// Mitsubishi GX Works2 project: group10   PLC: FX3G

// global labels: Global1
VAR_GLOBAL
  EmergencyEnd AT X005 : BOOL;
  EndDay AT M7 : BOOL;
  MaterialMissing AT M6 : BOOL;
  WorkDayActive AT Y007 : BOOL;
  PrepStart AT X001 : BOOL;
  AnalogInput1 AT D8280 : INT;
  FloatInput AT D6000 : REAL;
END_VAR
VAR_GLOBAL CONSTANT
  Constant400 : REAL := E400.0;
END_VAR
VAR_GLOBAL
  TypeValue AT D1900 : REAL;
END_VAR
VAR_GLOBAL CONSTANT
  Const6 : REAL := 6.0;
END_VAR
VAR_GLOBAL
  Pinuk AT M2 : BOOL;
END_VAR
VAR_GLOBAL CONSTANT
  Const5 : REAL := 5.0;
END_VAR
VAR_GLOBAL
  Ragil AT M3 : BOOL;
  KeepPinuk AT M10 : BOOL;
  KeepRagil AT M12 : BOOL;
  InputRaspberryAmount AT D1500 : REAL;
  RaspberryAmount AT D1510 : REAL;
  InputLemonAmount AT D1600 : REAL;
  LemonAmount AT D1610 : REAL;
  InputMaterialAmount AT D1700 : REAL;
  MaterialAmount AT D1710 : REAL;
  InputGummyAmount AT D1800 : REAL;
  GummyAmount AT D1810 : REAL;
END_VAR
VAR_GLOBAL CONSTANT
  MinRaspberryPinuk : REAL := 385.0;
  MinLemonPinuk : REAL := 665.0;
  MinMaterialPinuk : REAL := 210.0;
  MinGummyPinuk : REAL := 70.0;
END_VAR
VAR_GLOBAL
  CantMakePinuk AT M13 : BOOL;
END_VAR
VAR_GLOBAL CONSTANT
  MinRaspberryRagil : REAL := 280.0;
  MinLemonRagil : REAL := 455;
  MinMaterialRagil : REAL := 105;
  MinGummyRagil : REAL := 28;
END_VAR
VAR_GLOBAL
  CantMakeRagil AT M14 : BOOL;
  StartWorkDay AT X007 : BOOL;
  Invalid AT M77 : BOOL;
  StartMaking AT M8 : BOOL;
END_VAR
VAR_GLOBAL CONSTANT
  Const0 : REAL := E0.0;
  Const700 : REAL := E700.0;
END_VAR
VAR_GLOBAL
  ContainerMR AT D1400 : REAL;
END_VAR
VAR_GLOBAL CONSTANT
  Const560 : REAL := E560.0;
END_VAR
VAR_GLOBAL
  ContainerML AT D1300 : REAL;
END_VAR
VAR_GLOBAL CONSTANT
  Const490 : REAL := E490.0;
  Const350 : REAL := E350.0;
END_VAR
VAR_GLOBAL
  HoldTime AT M9 : BOOL;
  TC_1 AT TC1 : BOOL;
END_VAR
VAR_GLOBAL CONSTANT
  Const5sec : INT := 50;
END_VAR
VAR_GLOBAL
  EndMakingLight AT TS1 : BOOL;
  Making AT Y000 : BOOL;
  Freezing AT X002 : BOOL;
  TempS AT X003 : BOOL;
  FinishFreezing AT TS2 : BOOL;
  FreezingLight AT Y002 : BOOL;
  TC_2 AT TC2 : BOOL;
END_VAR
VAR_GLOBAL CONSTANT
  Const8sec : INT := 80;
END_VAR
VAR_GLOBAL
  ContainerFL AT D1310 : REAL;
  ContainerFR AT D1410 : REAL;
  Mixing AT M15 : BOOL;
  ContainerMix AT D1955 : REAL;
  PinukMixed AT M20 : BOOL;
  RagilMixed AT M30 : BOOL;
  TimerMixPinuk AT TC10 : BOOL;
END_VAR
VAR_GLOBAL CONSTANT
  Mix5Sec : INT := 50;
END_VAR
VAR_GLOBAL
  StopMixPinuk AT TS10 : BOOL;
  FinishMixPinukLight AT M40 : BOOL;
  TimerMixRagil AT TC11 : BOOL;
END_VAR
VAR_GLOBAL CONSTANT
  Mix3Sec : INT := 30;
END_VAR
VAR_GLOBAL
  StopMixRagil AT TS11 : BOOL;
  FinishMixRagilLight AT M50 : BOOL;
  HelpFlick AT M60 : BOOL;
  TC_3 AT TC3 : BOOL;
  HelpFlick1 AT TS3 : BOOL;
  Flick1 AT Y005 : BOOL;
  TC_4 AT TC4 : BOOL;
  HelpFlick2 AT TS4 : BOOL;
  Flick2 AT Y006 : BOOL;
END_VAR
VAR_GLOBAL CONSTANT
  Const1Sec : INT := 10;
END_VAR
VAR_GLOBAL
  PackageAmount AT D1360 : REAL;
END_VAR
VAR_GLOBAL CONSTANT
  AddOnePackage : REAL := 1;
  Const40 : REAL := E40.0;
END_VAR
VAR_GLOBAL
  OutputP AT D1100 : REAL;
  AnalogOutput AT D8282 : INT;
  WaitToPack AT M90 : BOOL;
END_VAR

// task Task_01 (event TRUE, interval 0, priority 31): POU_01

PROGRAM POU_01
(* structured ladder/FBD written out as ST: instructions are called as NAME(EN, inputs, outputs); _pN, _eN, _tN stand for wires *)
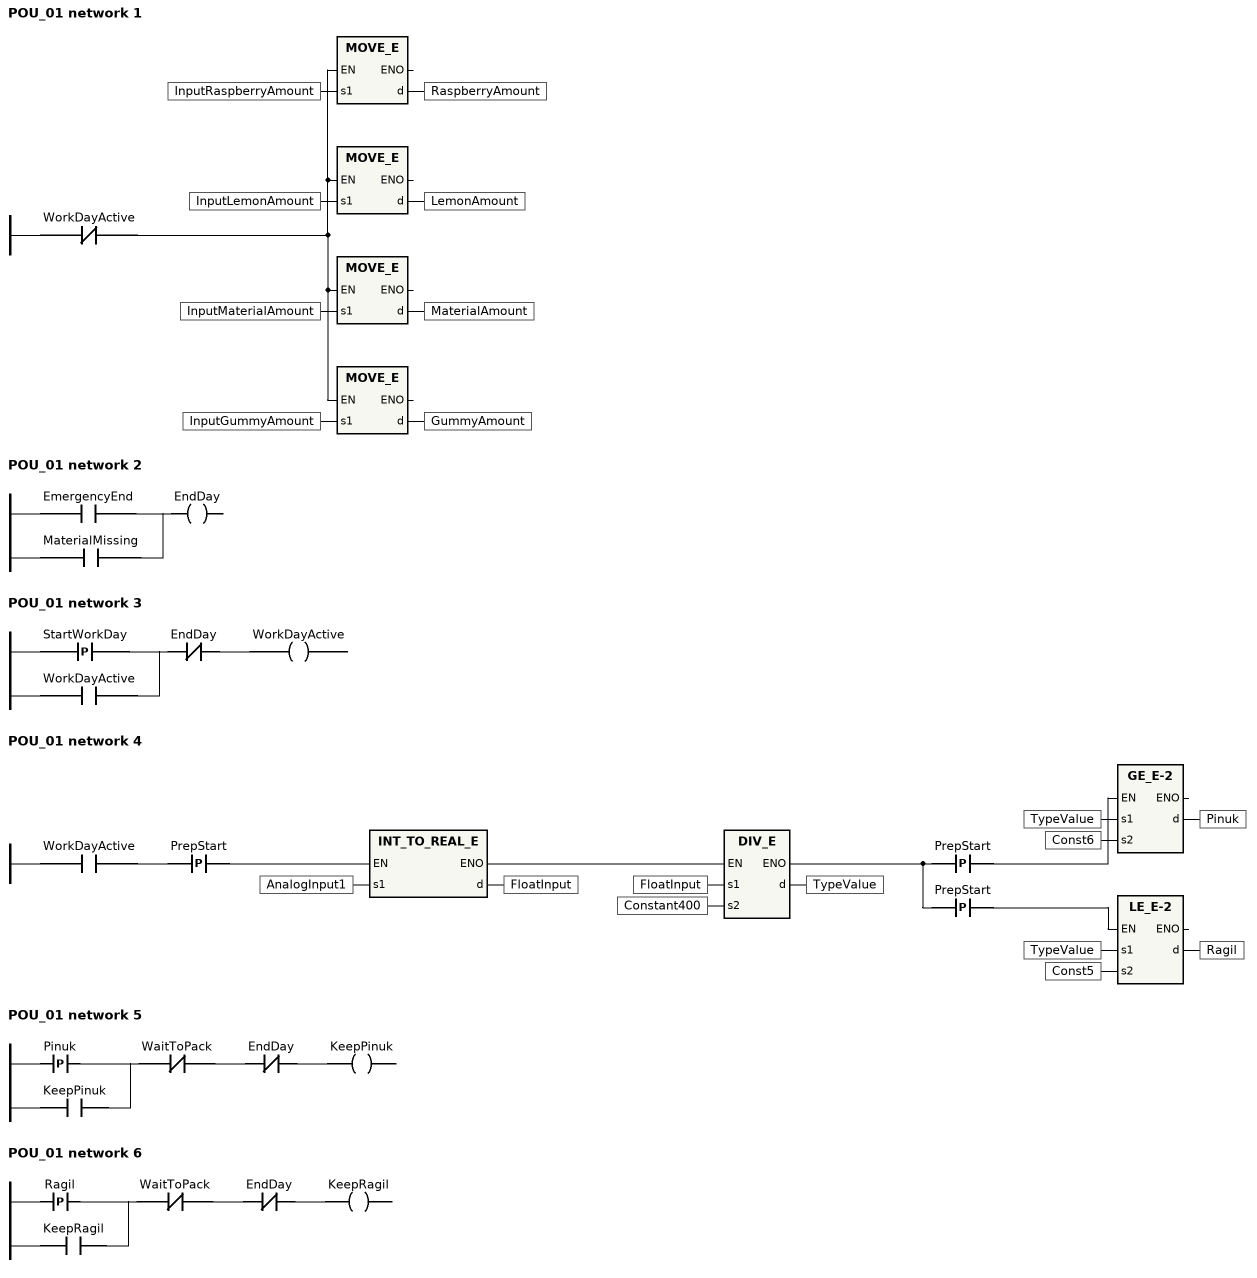
(* network 1 *)
_p1 := NOT WorkDayActive;
MOVE_E(_p1, InputRaspberryAmount, RaspberryAmount);
MOVE_E(_p1, InputLemonAmount, LemonAmount);
MOVE_E(_p1, InputMaterialAmount, MaterialAmount);
MOVE_E(_p1, InputGummyAmount, GummyAmount);
(* network 2 *)
EndDay := EmergencyEnd OR MaterialMissing;
(* network 3 *)
WorkDayActive := (LDP(TRUE, StartWorkDay) OR WorkDayActive) AND NOT EndDay;
(* network 4 *)
_e1 := INT_TO_REAL_E(WorkDayActive AND LDP(TRUE, PrepStart), AnalogInput1, FloatInput);
_e2 := DIV_E(_e1, FloatInput, Constant400, TypeValue);
GE_E(_e2 AND LDP(TRUE, PrepStart), TypeValue, Const6, Pinuk);
LE_E(_e2 AND LDP(TRUE, PrepStart), TypeValue, Const5, Ragil);
(* network 5 *)
KeepPinuk := ((LDP(TRUE, Pinuk) OR KeepPinuk) AND NOT WaitToPack) AND NOT EndDay;
(* network 6 *)
KeepRagil := ((LDP(TRUE, Ragil) OR KeepRagil) AND NOT WaitToPack) AND NOT EndDay;
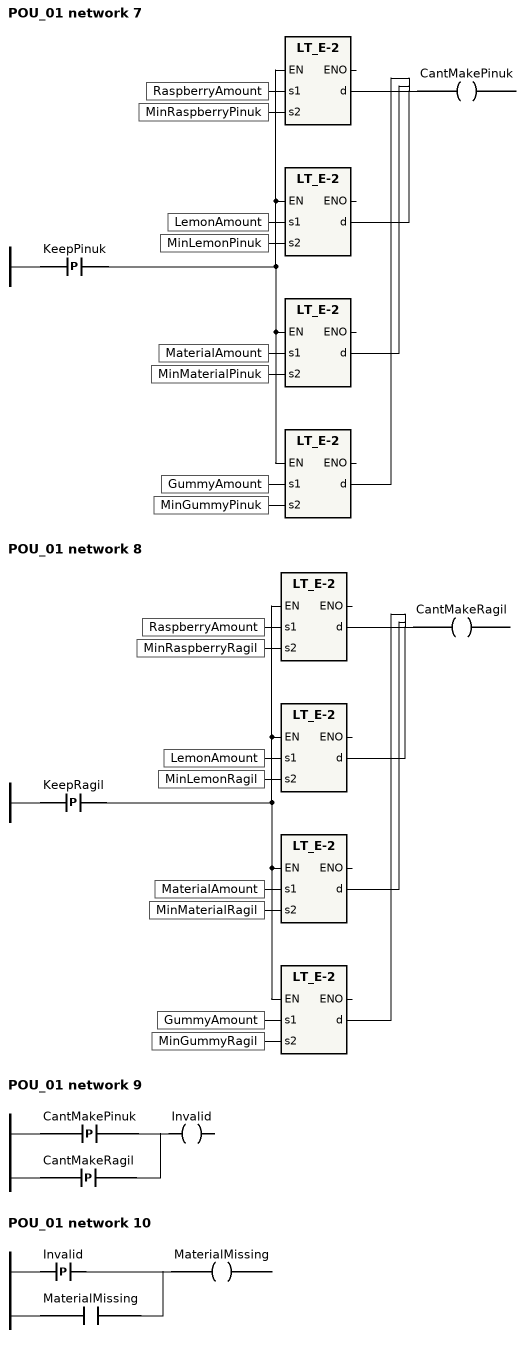
(* network 7 *)
_p1 := LDP(TRUE, KeepPinuk);
LT_E(_p1, RaspberryAmount, MinRaspberryPinuk, _t2);
LT_E(_p1, LemonAmount, MinLemonPinuk, _t3);
LT_E(_p1, MaterialAmount, MinMaterialPinuk, _t4);
LT_E(_p1, GummyAmount, MinGummyPinuk, _t5);
CantMakePinuk := _t2 OR _t3 OR _t4 OR _t5;
(* network 8 *)
_p1 := LDP(TRUE, KeepRagil);
LT_E(_p1, RaspberryAmount, MinRaspberryRagil, _t2);
LT_E(_p1, LemonAmount, MinLemonRagil, _t3);
LT_E(_p1, MaterialAmount, MinMaterialRagil, _t4);
LT_E(_p1, GummyAmount, MinGummyRagil, _t5);
CantMakeRagil := _t2 OR _t3 OR _t4 OR _t5;
(* network 9 *)
Invalid := LDP(TRUE, CantMakePinuk) OR LDP(TRUE, CantMakeRagil);
(* network 10 *)
MaterialMissing := LDP(TRUE, Invalid) OR MaterialMissing;
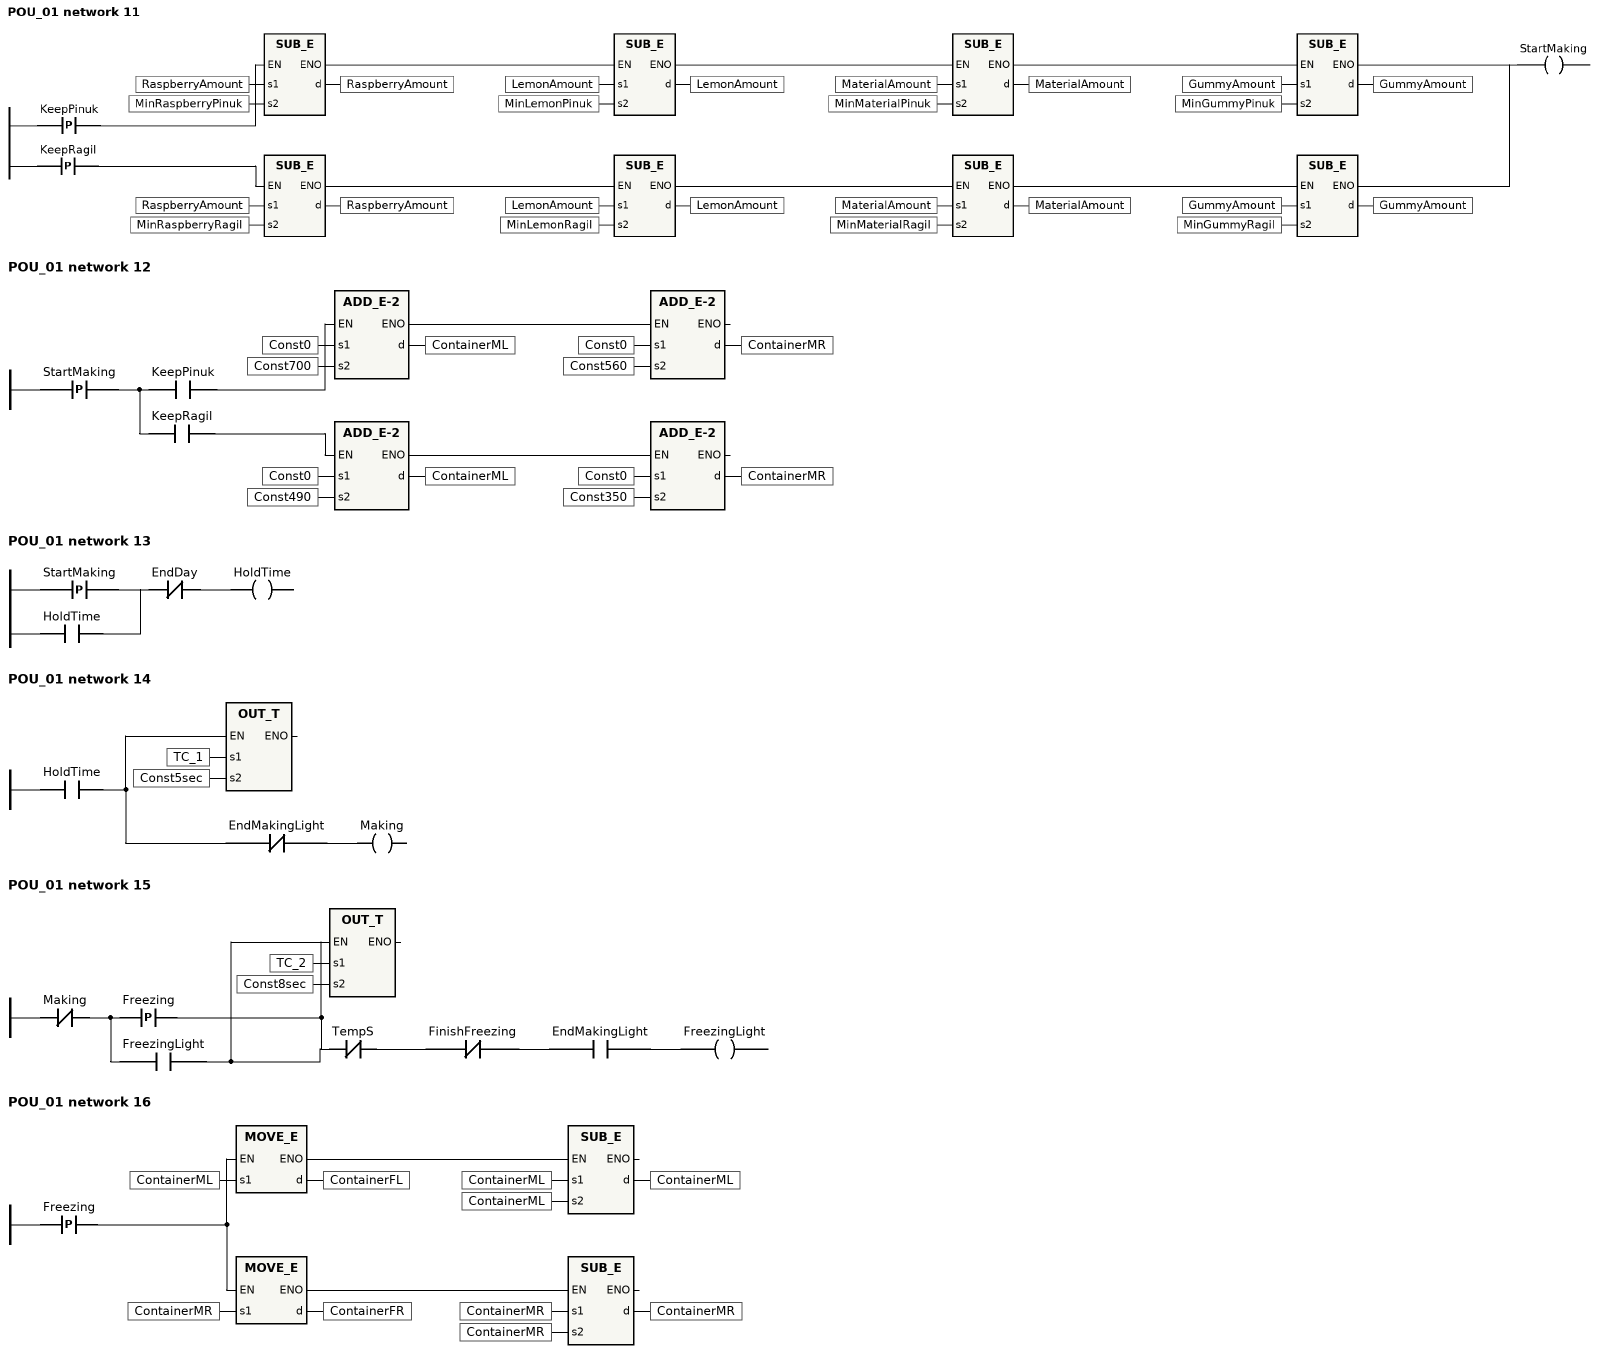
(* network 11 *)
_e1 := SUB_E(LDP(TRUE, KeepPinuk), RaspberryAmount, MinRaspberryPinuk, RaspberryAmount);
_e2 := SUB_E(_e1, LemonAmount, MinLemonPinuk, LemonAmount);
_e3 := SUB_E(_e2, MaterialAmount, MinMaterialPinuk, MaterialAmount);
_e4 := SUB_E(_e3, GummyAmount, MinGummyPinuk, GummyAmount);
_e5 := SUB_E(LDP(TRUE, KeepRagil), RaspberryAmount, MinRaspberryRagil, RaspberryAmount);
_e6 := SUB_E(_e5, LemonAmount, MinLemonRagil, LemonAmount);
_e7 := SUB_E(_e6, MaterialAmount, MinMaterialRagil, MaterialAmount);
_e8 := SUB_E(_e7, GummyAmount, MinGummyRagil, GummyAmount);
StartMaking := _e4 OR _e8;
(* network 12 *)
_p1 := LDP(TRUE, StartMaking);
_e2 := ADD_E(_p1 AND KeepPinuk, Const0, Const700, ContainerML);
ADD_E(_e2, Const0, Const560, ContainerMR);
_e3 := ADD_E(_p1 AND KeepRagil, Const0, Const490, ContainerML);
ADD_E(_e3, Const0, Const350, ContainerMR);
(* network 13 *)
HoldTime := (LDP(TRUE, StartMaking) OR HoldTime) AND NOT EndDay;
(* network 14 *)
OUT_T(HoldTime, TC_1, Const5sec);
Making := HoldTime AND NOT EndMakingLight;
(* network 15 *)
_p1 := NOT Making;
_p2 := (_p1 AND LDP(TRUE, Freezing)) OR (_p1 AND FreezingLight);
OUT_T(_p2, TC_2, Const8sec);
FreezingLight := _p2 AND NOT TempS AND NOT FinishFreezing AND EndMakingLight;
(* network 16 *)
_p1 := LDP(TRUE, Freezing);
_e2 := MOVE_E(_p1, ContainerML, ContainerFL);
SUB_E(_e2, ContainerML, ContainerML, ContainerML);
_e3 := MOVE_E(_p1, ContainerMR, ContainerFR);
SUB_E(_e3, ContainerMR, ContainerMR, ContainerMR);
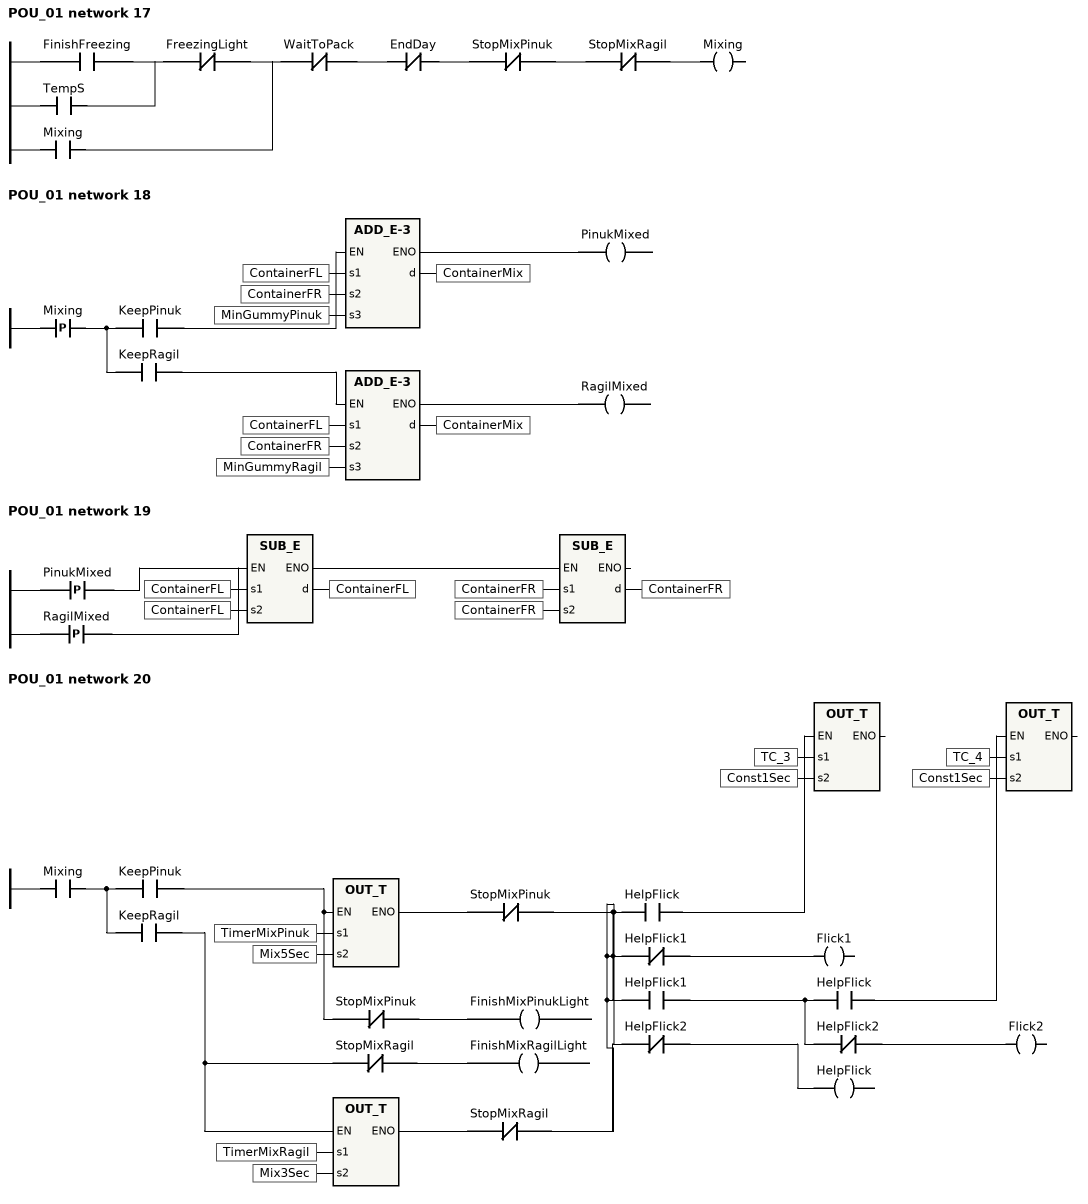
(* network 17 *)
Mixing := ((((((FinishFreezing OR TempS) AND NOT FreezingLight) OR Mixing) AND NOT WaitToPack) AND NOT EndDay) AND NOT StopMixPinuk) AND NOT StopMixRagil;
(* network 18 *)
_p1 := LDP(TRUE, Mixing);
_e2 := ADD_E(_p1 AND KeepPinuk, ContainerFL, ContainerFR, MinGummyPinuk, ContainerMix);
PinukMixed := _e2;
_e3 := ADD_E(_p1 AND KeepRagil, ContainerFL, ContainerFR, MinGummyRagil, ContainerMix);
RagilMixed := _e3;
(* network 19 *)
_e1 := SUB_E(LDP(TRUE, PinukMixed) OR LDP(TRUE, RagilMixed), ContainerFL, ContainerFL, ContainerFL);
SUB_E(_e1, ContainerFR, ContainerFR, ContainerFR);
(* network 20 *)
_p1 := Mixing AND KeepPinuk;
_e2 := OUT_T(_p1, TimerMixPinuk, Mix5Sec);
_p3 := Mixing AND KeepRagil;
_e4 := OUT_T(_p3, TimerMixRagil, Mix3Sec);
_p5 := (_e2 AND NOT StopMixPinuk) OR (_e4 AND NOT StopMixRagil);
OUT_T(_p5 AND HelpFlick, TC_3, Const1Sec);
FinishMixPinukLight := _p1 AND NOT StopMixPinuk;
Flick1 := _p5 AND NOT HelpFlick1;
_p6 := _p5 AND HelpFlick1;
OUT_T(_p6 AND HelpFlick, TC_4, Const1Sec);
Flick2 := _p6 AND NOT HelpFlick2;
FinishMixRagilLight := _p3 AND NOT StopMixRagil;
HelpFlick := _p5 AND NOT HelpFlick2;
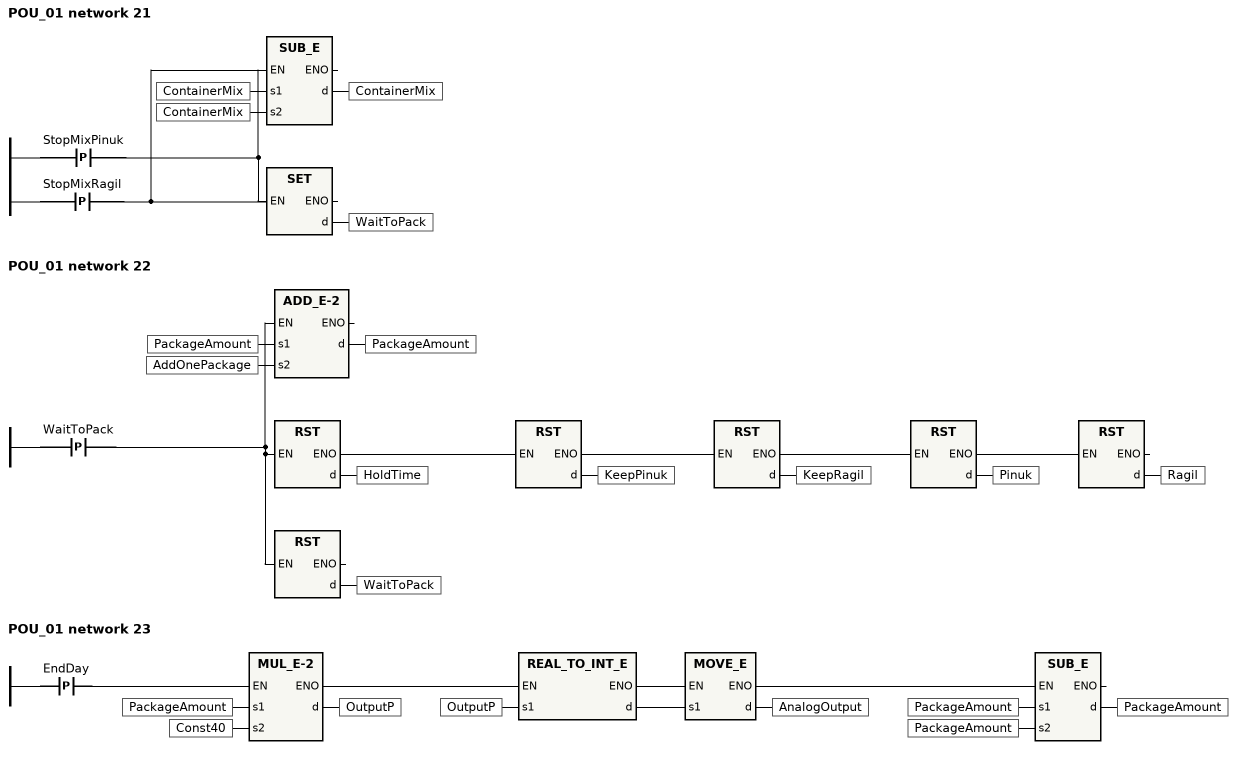
(* network 21 *)
_p1 := LDP(TRUE, StopMixPinuk) OR LDP(TRUE, StopMixRagil);
SUB_E(_p1, ContainerMix, ContainerMix, ContainerMix);
SET(_p1, WaitToPack);
(* network 22 *)
_p1 := LDP(TRUE, WaitToPack);
ADD_E(_p1, PackageAmount, AddOnePackage, PackageAmount);
_e2 := RST(_p1, HoldTime);
_e3 := RST(_e2, KeepPinuk);
_e4 := RST(_e3, KeepRagil);
_e5 := RST(_e4, Pinuk);
RST(_e5, Ragil);
RST(_p1, WaitToPack);
(* network 23 *)
_e1 := MUL_E(LDP(TRUE, EndDay), PackageAmount, Const40, OutputP);
_e3 := REAL_TO_INT_E(_e1, OutputP, _t2);
_e4 := MOVE_E(_e3, _t2, AnalogOutput);
SUB_E(_e4, PackageAmount, PackageAmount, PackageAmount);
END_PROGRAM
